RoboDK station: Claude.rdk

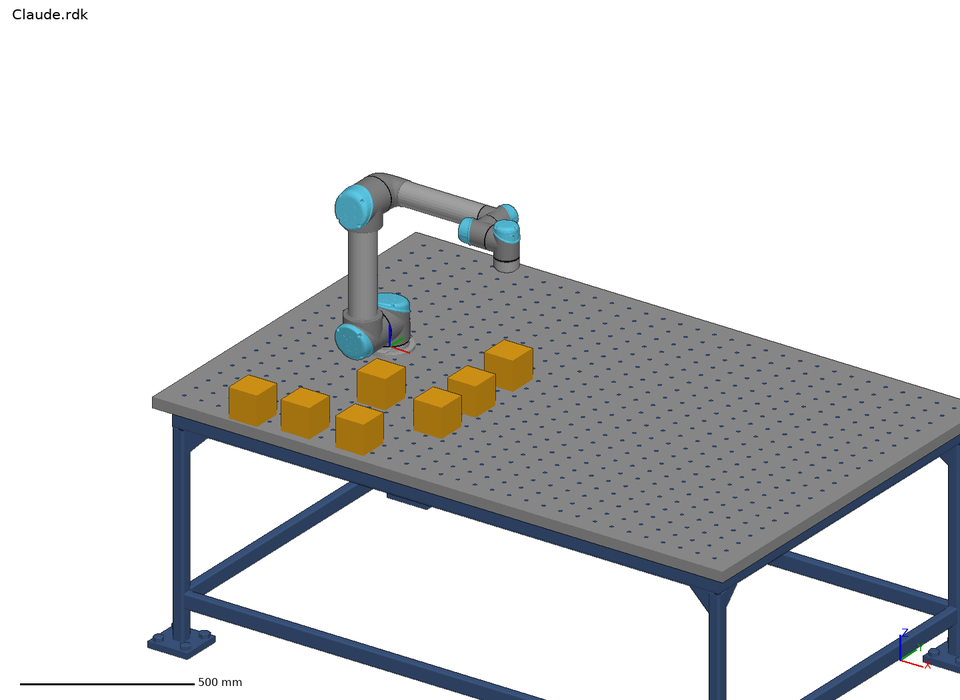
[picture v0: the station drawn from its stored meshes, robots at their saved joint values, targets as dots, program paths as lines]
Station Claude (saved by RoboDK 5.5.4). Poses are relative to the parent item; angles as X-Y-Z fixed-axis rotations.
  - object Table at (0, 0, 0) mm, size 2020 x 1340 x 800 mm, geometry from Table-2000mmx1200mmx800mm.sld
  - object Cube1 at (360, 60, 0) mm, rotated rx 0 ry 0 rz -90 deg, size 100 x 100 x 100 mm, geometry from Cube-100mm.sld
  - object Cube2 at (370, -140, 0) mm, rotated rx 0 ry 0 rz -90 deg, size 100 x 100 x 100 mm, geometry from Cube-100mm.sld
  - object Cube3 at (370, -310, 0) mm, rotated rx 0 ry 0 rz -90 deg, size 100 x 100 x 100 mm, geometry from Cube-100mm.sld
  - object Cube4 at (130, -250, 0) mm, rotated rx 0 ry 0 rz -90 deg, size 100 x 100 x 100 mm, geometry from Cube-100mm.sld
  - object Cube5 at (250, -530, 0) mm, rotated rx 0 ry 0 rz -90 deg, size 100 x 100 x 100 mm, geometry from Cube-100mm.sld
  - object Cube6 at (60, -530, 0) mm, rotated rx 0 ry 0 rz -90 deg, size 100 x 100 x 100 mm, geometry from Cube-100mm.sld
  - object Cube7 at (-110, -550, 0) mm, rotated rx 0 ry 0 rz -90 deg, size 100 x 100 x 100 mm, geometry from Cube-100mm.sld
  - frame UR5 Base at (0, 0, 0) mm
    - robot UR5: 6 axes
        modified DH rows (alpha deg, a mm, theta deg, d mm): 0, 0, 0, 89.2; 90, 0, 180, 0; 0, 425, 0, 0; 0, 392, 0, 109.3; -90, 0, 0, 94.75; 90, 0, 180, 82.5
        joint limits [-360, -360, -360, -360, -360, -360] to [360, 360, 360, 360, 360, 360]; home [0, -90, -90, 0, 90, 0]; saved at [0, -90, -90, -90, 90, 0]
